// Mitsubishi GX Works2 project: BKVinaMainV1   PLC: FX3U/FX3UC

// global labels: Global1
VAR_GLOBAL
  RelayMXDT_1 AT Y002 : BOOL;
  RelayMXDT_2 AT Y006 : BOOL;
  RelayMXDP_1 AT Y003 : BOOL;
  RelayMXDP_2 AT Y007 : BOOL;
  RelayMQ_R AT Y010 : BOOL;
  MR_DSLOW AT Y011 : BOOL;
  RelayMR_1 AT Y012 : BOOL;
  RelayMR_2 AT Y013 : BOOL;
  RelayTT AT Y014 : BOOL;
  ALARM AT Y015 : BOOL;
  OPERATION AT Y016 : BOOL;
  RelayXLKC1 AT Y017 : BOOL;
  RelayXLC2 AT Y020 : BOOL;
  RelayXLD3_1 AT Y021 : BOOL;
  RelayXLD3_2 AT Y022 : BOOL;
  RelayXLX4_1 AT Y023 : BOOL;
  RelayXLX4_2 AT Y024 : BOOL;
  RelayXLX5_1 AT Y025 : BOOL;
  RelayXLX5_2 AT Y026 : BOOL;
  RelayXLD6_1 AT Y027 : BOOL;
  RelayXLD6_2 AT Y030 : BOOL;
  RelayXLTT AT Y031 : BOOL;
  RelayXLTP AT Y032 : BOOL;
  RelayXLKDT AT Y035 : BOOL;
  RelayLubOil AT Y036 : BOOL;
  RelayOilP AT Y037 : BOOL;
  RelayOilV1 AT Y040 : BOOL;
  RelayOilV2 AT Y041 : BOOL;
  CommandMXC_F : BOOL;
  CommandMXC_Z : BOOL;
  CommandMQ_F : BOOL;
  CommandMQ_Z : BOOL;
  CommandMXDT_F : BOOL;
  CommandMXDT_Z : BOOL;
  CommandMXDP_F : BOOL;
  CommandMXDP_Z : BOOL;
  CommandMR_L : BOOL;
  CommandMR_R : BOOL;
  CommandXLXC_I : BOOL;
  CommandXLXC_O : BOOL;
  MR_L AT X010 : BOOL;
  MR_R AT X011 : BOOL;
  CB3 AT X012 : BOOL;
  EMERG AT X013 : BOOL;
  MainRST AT X014 : BOOL;
  START AT X015 : BOOL;
  Jog_Left AT X016 : BOOL;
  Jog_Right AT X017 : BOOL;
  PushOilPump AT X020 : BOOL;
  XLKC1_I AT X021 : BOOL;
  XLKC1_O AT X022 : BOOL;
  XLC2_I AT X023 : BOOL;
  XLC2_O AT X024 : BOOL;
  XLD3_I AT X025 : BOOL;
  XLD3_O AT X026 : BOOL;
  XLX4_I AT X027 : BOOL;
  XLX4_O AT X030 : BOOL;
  XLX5_I AT X031 : BOOL;
  XLX5_O AT X032 : BOOL;
  XLD6_I AT X033 : BOOL;
  XLD6_O AT X034 : BOOL;
  XLTT_I AT X035 : BOOL;
  XLTP_I AT X036 : BOOL;
  XLTT_O AT X037 : BOOL;
  XLTP_O AT X040 : BOOL;
  XLDT_I AT X041 : BOOL;
  XLDT_O AT X042 : BOOL;
  XLDP_I AT X043 : BOOL;
  XLDP_O AT X044 : BOOL;
  OLPump AT X045 : BOOL;
  MR_L1 AT X046 : BOOL;
  MR_R1 AT X047 : BOOL;
  RelayMQ_2 AT Y005 : BOOL;
  RelayMXC_1 AT Y000 : BOOL;
  RelayMXC_2 AT Y004 : BOOL;
  RelayMQ_1 AT Y001 : BOOL;
  MXDT_ZX AT X002 : BOOL;
  MXDP_ZX AT X003 : BOOL;
  MXC_ZX AT X004 : BOOL;
  MQ_ZX AT X005 : BOOL;
  MXC_FWD : BOOL;
  MQ_FWD : BOOL;
  MXDT_FWD : BOOL;
  MXDP_FWD : BOOL;
  ModeAuto : BOOL;
  StopEmerg : BOOL;
  activeCK : BOOL;
  pushManXLKC1 AT M200 : BOOL;
  pushManXLC2 AT M201 : BOOL;
  pushManXLD3_I AT M202 : BOOL;
  pushManXLD3_O AT M203 : BOOL;
  pushManXLX4_I AT M204 : BOOL;
  pushManXLX4_O AT M205 : BOOL;
  pushManXLX5_I AT M206 : BOOL;
  pushManXLX5_O AT M207 : BOOL;
  pushManXLD6_I AT M208 : BOOL;
  pushManXLD6_O AT M209 : BOOL;
  pushManXLTT AT M210 : BOOL;
  pushManXLTP AT M211 : BOOL;
  pushManXLKDT AT M212 : BOOL;
  pushManXLKDP AT M213 : BOOL;
  pushManXLDT AT M214 : BOOL;
  pushManXLDP AT M215 : BOOL;
  pushManTT AT M216 : BOOL;
  pushManMXC_F AT M217 : BOOL;
  pushManMXC_Z AT M218 : BOOL;
  pushManMQ_F AT M219 : BOOL;
  pushManMQ_Z AT M220 : BOOL;
  pushManMXDT_F AT M221 : BOOL;
  pushManMXDT_Z AT M222 : BOOL;
  pushManMXDP_F AT M223 : BOOL;
  pushManMXDP_Z AT M224 : BOOL;
  PushOilV1 AT M225 : BOOL;
  PushOilV2 AT M226 : BOOL;
  pushB8 AT M227 : BOOL;
  pushB9 AT M228 : BOOL;
  pushB10 AT M229 : BOOL;
  pushCa1 AT M230 : BOOL;
  pushCa2 AT M231 : BOOL;
  pushCa3 AT M232 : BOOL;
  rstTotalB AT M233 : BOOL;
  rstCounterCK AT M234 : BOOL;
  rstAmountCK AT M235 : BOOL;
  restory AT M236 : BOOL;
  PushLubOil AT M237 : BOOL;
  PushPause AT M238 : BOOL;
  Pape0 AT M239 : BOOL;
  Pape1 AT M240 : BOOL;
  Pape2 AT M241 : BOOL;
  Pape3 AT M242 : BOOL;
  CommandXLX5_I : BOOL;
  CommandXLX5_O : BOOL;
  CommandXLXD_I : BOOL;
  CommandXLXD_O : BOOL;
  CommandXLD6_I : BOOL;
  PauseAlarm AT M243 : BOOL;
  RelayXLDT AT Y033 : BOOL;
  RelayXLDP AT Y034 : BOOL;
  PauseMR AT M244 : BOOL;
  Real_MXC : REAL;
  Real_MQ : REAL;
  Real_MXDT : REAL;
  Real_MXDP : REAL;
  Counter_MQ : DINT;
  Round_MXC AT D200 : REAL;
  Round_MQL AT D202 : REAL;
  Round_MQR AT D204 : REAL;
  Round_MXDT AT D206 : REAL;
  Round_MXDP AT D208 : REAL;
  IndicateMXC AT D210 : REAL;
  IndicateMQ AT D212 : REAL;
  IndicateMXDT AT D214 : REAL;
  IndicateMXDP AT D216 : REAL;
  NumberCK AT D220 : DWORD;
  CounterCK AT D222 : DWORD;
  AmountCK AT D224 : DWORD;
  TotalCK AT D226 : DWORD;
  rstPauseMR AT M245 : BOOL;
  ca1_B8 AT D250 : DWORD;
  ca2_B8 AT D252 : DWORD;
  ca3_B8 AT D254 : DWORD;
  ca1_B9 AT D256 : DWORD;
  ca2_B9 AT D258 : DWORD;
  ca3_B9 AT D260 : DWORD;
  ca1_B10 AT D262 : DWORD;
  ca2_B10 AT D264 : DWORD;
  ca3_B10 AT D266 : DWORD;
  total_B8 AT D268 : DWORD;
  total_B9 AT D270 : DWORD;
  total_B10 AT D272 : DWORD;
  CommandMXDT : BOOL;
  CommandMXDP : BOOL;
  CommandBTX : BOOL;
  CommandXLTT : BOOL;
  CommandXLTP : BOOL;
  CommandXLDT : BOOL;
  CommandXLDP : BOOL;
  CommandXLKDT : BOOL;
  CommandXLKDP : BOOL;
  CommandXLKC1 : BOOL;
  MXC_Z : BOOL;
  MQ_Z : BOOL;
  MXDT_Z : BOOL;
  MXDP_Z : BOOL;
  MQ_LimitF : BOOL;
  MQ_LimitR : BOOL;
  CommandXLD6_O : BOOL;
  TimeMR_DSL AT D230 : DWORD;
  TimeMQ_Z AT D232 : DWORD;
  TimeMR_E AT D234 : DWORD;
  TimeERROR AT D236 : DWORD;
  TimeMXD AT D238 : DWORD;
END_VAR

// task InterruptMQ_Z (event I501, interval 0, priority 31): PickupX005
// task InterruptMXC (event I010, interval 0, priority 31): EncoderX001
// task InterruptMXC_Z (event I401, interval 0, priority 31): PickupX004
// task InterruptMXDP (event I030, interval 0, priority 31): EncoderX007
// task InterruptMXDP_Z (event I301, interval 0, priority 31): PickupX003
// task InterruptMXDT (event I020, interval 0, priority 31): EncoderX006
// task InterruptMXDT_Z (event I201, interval 0, priority 31): PickupX002
// task Task_01 (event TRUE, interval 0, priority 31): PowerControl, StepControl

PROGRAM EncoderX001
SET( TRUE , MXC_FWD );
SET( TRUE, CommandMXC_Z);
RST( TRUE, CommandXLXC_O);
RST( TRUE, CommandXLXD_O);
END_PROGRAM

PROGRAM EncoderX006
SET( TRUE , MXDT_FWD );
RST( TRUE, CommandXLDT);
RST( TRUE, CommandMXDT_F);
RST( TRUE, CommandMXDT);
SET( XLX4_O AND activeCK, CommandXLXC_I); 
SET( XLD3_O AND activeCK, CommandXLXD_I);
END_PROGRAM

PROGRAM EncoderX007
SET( TRUE , MXDP_FWD );
RST( TRUE, CommandXLDP);
RST( TRUE, CommandMXDP_F);
RST( TRUE, CommandMXDP);
END_PROGRAM

FUNCTION_BLOCK MotorOne
VAR_INPUT
  SetAutoMan : BOOL;
  PushMan : BOOL;
  LimitInput : BOOL;
END_VAR
VAR_IN_OUT
  SetAutoRun : BOOL;
END_VAR
VAR_OUTPUT
  Output : BOOL;
END_VAR
VAR
  RelayBuffer : BOOL;
END_VAR
(* Set mode Auto / Mannual *)
IF  SetAutoMan THEN
	RelayBuffer := SetAutoRun;
ELSE 
	RelayBuffer := PushMan;
END_IF;

Output := RelayBuffer AND NOT LimitInput ;
(* Reset control signal *)
RST(LDP(TRUE, LimitInput), SetAutoRun );
END_FUNCTION_BLOCK

FUNCTION_BLOCK MotorRev
VAR_INPUT
  SetAutoMan : BOOL;
END_VAR
VAR_IN_OUT
  PushManF : BOOL;
  PushManR : BOOL;
END_VAR
VAR_INPUT
  LimitInputF : BOOL;
  LimitInputR : BOOL;
END_VAR
VAR_IN_OUT
  SetAutoRunF : BOOL;
  SetAutoRunR : BOOL;
END_VAR
VAR_OUTPUT
  OutputF : BOOL;
  OutputR : BOOL;
END_VAR
VAR
  RelayBufferF : BOOL;
  RelayBufferR : BOOL;
END_VAR
(* Set mode Auto/Man *)
IF  SetAutoMan THEN
	RelayBufferF := 	NOT SetAutoRunR AND SetAutoRunF;
	RelayBufferR := NOT SetAutoRunF AND SetAutoRunR;
ELSE
	RelayBufferF := NOT PushManR AND PushManF;
	RelayBufferR := NOT PushManF AND PushManR;
END_IF;

OutputF := RelayBufferF AND NOT LimitInputF ;
OutputR := RelayBufferR AND NOT LimitInputR ;
(* Reset control signal *)
RST( LDP(TRUE, LimitInputF), SetAutoRunF );
RST( LDP(TRUE, LimitInputR), SetAutoRunR );
END_FUNCTION_BLOCK

PROGRAM PickupX002
SET(TRUE, MXDT_Z);
SET( TRUE, M8052);
RST( TRUE, CommandMXDT);
END_PROGRAM

PROGRAM PickupX003
SET(TRUE, MXDP_Z);
SET( TRUE, M8053);
RST( TRUE, CommandMXDP);
END_PROGRAM

PROGRAM PickupX004
SET( TRUE, MXC_Z);
SET( XLD3_O, CommandXLXD_I);
SET( XLX4_O, CommandXLXC_I);
SET( TRUE, M8054);
END_PROGRAM

PROGRAM PickupX005
DADD( MQ_LimitF, Counter_MQ, K1 , Counter_MQ);
SET( Counter_MQ >= REAL_TO_DINT( Real_MQ), MQ_FWD);
SET( MQ_LimitR , MQ_Z);
END_PROGRAM

PROGRAM PowerControl
VAR
  MR : MotorRev;
  MQ : MotorRev;
  MXC : MotorRev;
  MXDT : MotorRev;
  MXDP : MotorRev;
  XLKC1 : MotorOne;
  XLC2 : MotorOne;
  XLD3 : MotorRev;
  XLX4 : MotorRev;
  XLX5 : MotorRev;
  XLD6 : MotorRev;
  XLTT : MotorOne;
  XLTP : MotorOne;
  XLKDT : MotorOne;
  XLKDP : MotorOne;
  XLDT : MotorOne;
  XLDP : MotorOne;
  OILPUMP : MotorOne;
  VALVE1 : MotorOne;
  VALVE2 : MotorOne;
  ManualMXC_F : BOOL;
  ManualMXC_Z : BOOL;
  ManualMQ_F : BOOL;
  ManualMQ_Z : BOOL;
  ManualMXDT_F : BOOL;
  ManualMXDT_Z : BOOL;
  ManualMXDP_F : BOOL;
  ManualMXDP_Z : BOOL;
  CommandXLC2 : BOOL;
  ButtonOilP : BOOL;
  ButtonOilV1 : BOOL;
  ButtonOilV2 : BOOL;
  TimerMRDSL_Q : BOOL;
  TimerMQ_ZQ : BOOL;
  TimerMR_DSL : TON;
  TimerMQ_Z : TON;
  Dint_C251 : DINT;
  Dint_C234 : DINT;
  Dint_C244 : DINT;
  Dint_C245 : DINT;
  ManualXLD6 : BOOL;
  ManualXLDT : BOOL;
  ManualXLDP : BOOL;
  ManualXLKDT : BOOL;
  ManualXLKDP : BOOL;
  ManualXLX5_O : BOOL;
  ManualXLX5_I : BOOL;
  TimerXLTT : TON;
  TimerXLTP : TON;
  TimerXLTT_Q : BOOL;
  TimerXLTP_Q : BOOL;
END_VAR
EI( TRUE );
(* MR: Chạy khi cụm xoắn đầu chạy *)
MR(SetAutoMan := ModeAuto, PushManF := Jog_Left , PushManR := Jog_Right ,
		LimitInputF := MR_L, LimitInputR := MR_R,
		SetAutoRunF := CommandMR_L, SetAutoRunR := CommandMR_R ,
		OutputF := RelayMR_1, OutputR:= RelayMR_2);

RelayTT := (RelayMR_1 AND NOT MR_L) OR (RelayMR_2 AND NOT MR_R);
TimerMR_DSL(IN := (NOT MR_L AND RelayMR_1) OR (NOT MR_R AND RelayMR_2), 
								PT := DWORD_TO_TIME(TimeMR_DSL)/100, Q := TimerMRDSL_Q );
								
SET(LDP(TRUE, (MR_L1 AND RelayMR_1) OR (MR_R1 AND RelayMR_2)), MR_DSLOW);
RST(LDP(TRUE, (MR_L AND RelayMR_2) OR (MR_R AND RelayMR_1)), MR_DSLOW);

(* MXQ: *)	
SET(LDP(TRUE, MR_L OR MR_R), CommandMQ_F);
SET(LDP(TRUE, MR_L), RelayMQ_R);
RST(LDP(TRUE,MR_R), RelayMQ_R);
MQ(SetAutoMan := ModeAuto,
		PushManF := pushManMQ_F, PushManR := ManualMQ_Z,
		LimitInputF := MQ_FWD, LimitInputR := MQ_Z,
		SetAutoRunF := CommandMQ_F, SetAutoRunR := CommandMQ_Z, 
		OutputF := MQ_LimitF, OutputR:= MQ_LimitR);

IF RelayMQ_R THEN
	RelayMQ_1 := MQ_LimitF;
	RelayMQ_2 := MQ_LimitR;
ELSE
	RelayMQ_1 := MQ_LimitR;
	RelayMQ_2 := MQ_LimitF;
END_IF;
	
(* MXC:  CommandXLXC_I  and CommandXLXC_O *)	
MXC(SetAutoMan:= ModeAuto, 
			PushManF := pushManMXC_F, PushManR := ManualMXC_Z,
			LimitInputF := MXC_FWD, LimitInputR := MXC_Z,
			SetAutoRunF := CommandMXC_F, SetAutoRunR := CommandMXC_Z,
			OutputF := RelayMXC_1, OutputR := RelayMXC_2);

XLD3(SetAutoMan := ModeAuto,
			PushManF := pushManXLD3_O, PushManR := pushManXLD3_I,
			LimitInputF := XLD3_O, LimitInputR := XLD3_I,
			SetAutoRunF := CommandXLXD_O, SetAutoRunR := CommandXLXD_I,
			OutputF := RelayXLD3_1, OutputR := RelayXLD3_2);			
			
XLX4(SetAutoMan := ModeAuto,
			PushManF := pushManXLX4_O, PushManR := pushManXLX4_I,
			LimitInputF := XLX4_O , LimitInputR := XLX4_I,
			SetAutoRunF := CommandXLXC_O, SetAutoRunR := CommandXLXC_I,
			OutputF := RelayXLX4_1, OutputR := RelayXLX4_2);				

(* PHA:  CommandPHA_1  and CommandPHA_2 *)	
XLX5(SetAutoMan := ModeAuto,
			PushManF := pushManXLX5_O, PushManR := pushManXLX5_I,
			LimitInputF := NOT XLX4_I OR XLX5_O, LimitInputR := NOT XLX4_I OR XLX5_I,
			SetAutoRunF := CommandXLX5_O, SetAutoRunR := CommandXLX5_I,
			OutputF := RelayXLX5_1, OutputR := RelayXLX5_2);			

XLD6(SetAutoMan := ModeAuto,
			PushManF := pushManXLD6_O, PushManR := pushManXLD6_I,
			LimitInputF := FALSE, LimitInputR := FALSE,
			SetAutoRunF := CommandXLD6_O, SetAutoRunR := CommandXLD6_I, 
			OutputF := RelayXLD6_1, OutputR := RelayXLD6_2);				

(* MXDT:  CommandXLDT => dừng khi encoder đủ vòng *)	
SET( LDP(TRUE,  XLDT_I), CommandMXDT_Z);
MXDT(SetAutoMan := ModeAuto, 
			PushManF := pushManMXDT_F,  PushManR := ManualMXDT_Z,
			LimitInputF := MXDT_FWD, LimitInputR := MXDT_Z,
			SetAutoRunF :=  CommandMXDT_F, SetAutoRunR := CommandMXDT_Z ,
			OutputF := RelayMXDT_1, OutputR := RelayMXDT_2);

ManualXLDT := LDP(TRUE, pushManXLDT) XOR ManualXLDT;
RST( ModeAuto, ManualXLDT);
RelayXLDT := CommandXLDT OR ManualXLDT;

(* MXDP:  CommandXLDP => dừng khi encoder đủ vòng *)	
SET( LDP(TRUE, XLDP_I), CommandMXDP_Z);
MXDP(SetAutoMan := ModeAuto, 
			PushManF := pushManMXDP_F, PushManR := ManualMXDP_Z,
			LimitInputF := MXDP_FWD, LimitInputR := MXDP_Z,
			SetAutoRunF := CommandMXDP_F, SetAutoRunR := CommandMXDP_Z ,
			OutputF := RelayMXDP_1, OutputR := RelayMXDP_2);
			
ManualXLDP := LDP(TRUE, pushManXLDP) XOR ManualXLDP;
RST( ModeAuto, ManualXLDP);		
RelayXLDP := CommandXLDP OR ManualXLDP;

(* BTX:  CommandBTX  *)
RST(LDP(TRUE, CommandBTX AND XLKC1_O AND RelayXLKC1), CommandXLKC1);
SET(LDP(TRUE, CommandBTX AND XLC2_O AND RelayXLC2), CommandXLKC1);

RelayXLKC1 := (CommandXLKC1 AND ModeAuto) OR pushManXLKC1;

SET(LDP(TRUE, NOT XLKC1_O AND XLKC1_I), CommandXLC2);
RST(LDP(TRUE, NOT XLKC1_I AND XLKC1_O), CommandXLC2);
RST(LDP(TRUE, NOT XLKC1_I AND XLKC1_O), CommandBTX);

RelayXLC2 := (CommandXLC2 AND ModeAuto) OR pushManXLC2;

(* TLT: CommandXLTT => chạy theo cylinder  xoắn đầu *)
RelayXLTT := (RelayMXDT_1 AND ModeAuto) OR pushManXLTT;

(* TLP: CommandXLTP => chạy theo cylinder  xoắn đầu *)
RelayXLTP := (RelayMXDP_1 AND ModeAuto) OR pushManXLTP;

(* Hydrolic control *)
ButtonOilP := LDP(TRUE, PushOilPump) XOR ButtonOilP;
OILPUMP(PushMan := ButtonOilP, LimitInput := OLPump, Output := RelayOilP );

RelayOilV1 := RelayMQ_1 OR RelayMQ_2 OR RelayMXDP_1 OR RelayMXDP_2 
OR RelayMXDT_1 OR RelayMXDT_2 OR RelayXLX5_1 OR RelayXLX5_2;
RelayOilV2 := RelayMXC_1 OR RelayMXC_2 OR RelayXLD3_1 
OR RelayXLD3_2 OR RelayXLX4_1 OR RelayXLX4_2;
RelayLubOil := LDP(TRUE, PushLubOil) XOR RelayLubOil;

IF ModeAuto THEN
	(* Forward at Zero *)
	RST( CommandMXC_F AND MXC_ZX, MXC_FWD);
	RST( CommandMQ_F AND MQ_ZX, MQ_FWD);
	RST( CommandMXDT_F AND MXDT_ZX, MXDT_FWD);
	RST( CommandMXDP_F AND MXDP_ZX, MXDP_FWD);
	
	(* Set Home *)
	RST( LDP(TRUE, CommandMXC_Z), MXC_Z);
	RST( LDP(TRUE, CommandMQ_Z), MQ_Z);
	RST( LDP(TRUE, CommandMXDT_Z), MXDT_Z);
	RST( LDP(TRUE, CommandMXDP_Z), MXDP_Z);

ELSE	
	RST( LDP(TRUE, pushManMXC_F), MXC_FWD);
	RST( LDP(TRUE, pushManMQ_F), MQ_FWD);
	RST( LDP(TRUE, pushManMXDT_F), MXDT_FWD);
	RST( LDP(TRUE, pushManMXDP_F), MXDP_FWD);
	
	SET( LDP(TRUE, pushManMXC_Z), ManualMXC_Z);
	SET( LDP(TRUE, pushManMQ_Z), ManualMQ_Z);
	SET( LDP(TRUE, pushManMXDT_Z), ManualMXDT_Z);
	SET( LDP(TRUE, pushManMXDP_Z), ManualMXDP_Z);
	
	RST( LDP(TRUE, ManualMXC_Z), MXC_Z);
	RST( LDP(TRUE, ManualMQ_Z), MQ_Z);
	RST( LDP(TRUE, ManualMXDT_Z), MXDT_Z);
	RST( LDP(TRUE, ManualMXDP_Z), MXDP_Z);
	
	RST( LDP(TRUE, MXC_Z), ManualMXC_Z);
	RST( LDP(TRUE, MQ_Z), ManualMQ_Z);
	RST( LDP(TRUE, MXDT_Z), ManualMXDT_Z);
	RST( LDP(TRUE, MXDP_Z), ManualMXDP_Z);
	
	(* initialize encoder interrupt *)
	DMOVP( pushManMXC_F, 0, C251);
	DMOVP( pushManMQ_F, 0, Counter_MQ);
	DMOVP( pushManMXDT_F, 0, C244);
	DMOVP( pushManMXDP_F, 0, C245);
END_IF;

DWORD_TO_DINT_E( TRUE , C251 , Dint_C251 );
DWORD_TO_DINT_E( TRUE , C244 , Dint_C244 );
DWORD_TO_DINT_E( TRUE , C245 , Dint_C245 );

DEDIV( TRUE , DINT_TO_REAL(Dint_C251) , 2000.0 , IndicateMXC);
DEDIV( TRUE , DINT_TO_REAL(Counter_MQ) , 2.0 , IndicateMQ);
DEDIV( TRUE , DINT_TO_REAL(Dint_C244) , 360.0 , IndicateMXDT);
DEDIV( TRUE , DINT_TO_REAL(Dint_C245) , 360.0 , IndicateMXDP);

(* Set Interrupt *)
RST( LDP(TRUE, RelayMXC_2), M8054);
RST( RelayMQ_1 OR RelayMQ_2, M8055);
RST( LDP(TRUE, RelayMXDT_2), M8052);
RST( LDP(TRUE, RelayMXDP_2), M8053);

(* initialize encoder interrupt *)
DMOVP( CommandMXC_F, 0, C251);
DMOVP( CommandMQ_F, 0, Counter_MQ);
DMOVP( CommandMXDT_F, 0, C244);
DMOVP( CommandMXDP_F, 0, C245);

M8390 := M8388;
M8391 := M8388;
(*đảo chiều counter*)
M8244 := RelayMXDT_2;
M8245 := RelayMXDP_2;

(* Initialize high speed counter *)
OUT_C_32( TRUE, CC251, K2147483647);
OUT_C_32( TRUE, CC244, K2147483647);
OUT_C_32( TRUE, CC245, K2147483647);

(* Initialize high speed counter *)
DHSCS_I( TRUE , REAL_TO_DINT( Real_MXC ), CN251, I010);
DHSCS_I( TRUE , REAL_TO_DINT( Real_MXDT ), CN244, I020);
DHSCS_I( TRUE , REAL_TO_DINT( Real_MXDP ), CN245, I030);
END_PROGRAM

FUNCTION_BLOCK Servo
VAR_INPUT
  SetAutoMan : BOOL;
END_VAR
VAR_IN_OUT
  PushManF : BOOL;
  PushManR : BOOL;
END_VAR
VAR_INPUT
  Speed : DWORD;
  Range : DWORD;
END_VAR
VAR_IN_OUT
  SetAutoRunF : BOOL;
  SetAutoRunR : BOOL;
END_VAR
VAR_OUTPUT
  OutputPLS : BOOL;
  OutputDIR : BOOL;
END_VAR
VAR
  RelayPLS : BOOL;
  RelayDIR : BOOL;
END_VAR
VAR_INPUT
  LimitInputF : BOOL;
  LimitInputR : BOOL;
END_VAR
(* Set mode Auto/Man *)
IF  SetAutoMan THEN
	RelayDIR := SetAutoRunR;
	RelayPLS := SetAutoRunF XOR SetAutoRunR;
ELSE
	RelayDIR := PushManR;
	RelayPLS := PushManF XOR PushManR;
END_IF;

OutputDIR := RelayDIR ;

DPLSY( RelayPLS , Speed, Range , OutputPLS );

(* Reset control signal *)
RST( LDF( TRUE, LimitInputF ) , SetAutoRunF );
RST( LDF( TRUE, LimitInputR ) , SetAutoRunR );
END_FUNCTION_BLOCK

PROGRAM StepControl
VAR
  FistScan : BOOL;
  Emergency : BOOL;
  AutoEnable : BOOL;
  AuxCylinder : BOOL;
  MainCylinder : BOOL;
  TimerRestore : TON;
  TimerMR_E : TON;
  TimerERROR : TON;
  TimerMXDT : TON;
  TimerMXDP : TON;
  rstCa : BOOL;
  Error : ARRAY [0..18] OF BOOL;
  status : ARRAY [0..9] OF BOOL;
  cond : ARRAY [0..9] OF BOOL;
  count : INT;
  TimerMRR_Q : BOOL;
  TimerMRE_Q : BOOL;
  TimerERROR_Q : BOOL;
  TimerRestore_Q : BOOL;
  TimerMXDT_Q : BOOL;
  TimerMXDP_Q : BOOL;
  CylinderPha1 : BOOL;
  CylinderPha2 : BOOL;
  pointer : INT;
END_VAR
(*
Thake production line project: Mr. Chim Van Cang - Mr. Nguyen Tuan Nam
Code and graphic designer: HadiMadu - Techwaves Co,.Ltd
*)
Emergency := EMERG;

ALARM :=  NOT AutoEnable OR PauseAlarm;

SET(LDP(TRUE, MainRST), AutoEnable);
RST(LDP(TRUE, Emergency AND START), pointer);
SET(LDP(TRUE, Emergency AND START), status[0]);
RST(LDP(TRUE, Emergency AND START), AutoEnable);	

SET(LDP(TRUE, TimerMRE_Q), PauseMR);
RST(LDP(TRUE, rstPauseMR), PauseMR);

PauseAlarm := NOT CB3 OR PushPause OR PauseMR OR OLPump OR Emergency;(*OR TimerERROR_Q*)

OPERATION := status[1] OR status[2] OR status[3] OR status[4] OR status[5] OR status[6];
(* Mode Auto *)
ModeAuto := AutoEnable AND NOT PauseAlarm;

Pape0 := NOT ModeAuto;
Pape1 := status[0] OR status[1] OR status[2];
Pape2 := status[3] OR status[4];
Pape3 := status[5] OR status[6];

(* Power control *)
AuxCylinder := XLTT_I AND XLTP_I; 
MainCylinder := XLD3_I AND XLX4_I AND XLDT_I AND XLDP_I AND MQ_ZX;
CylinderPha1 := MR_L AND XLD6_O AND XLX5_I AND MXDT_ZX;
CylinderPha2 := MR_R AND XLD6_I AND XLX5_O AND MXDP_ZX;

cond[0] := pointer = 0 AND ModeAuto AND CylinderPha1 AND MainCylinder AND START; 			(* S1: Điều kiện chạy MQ*)
cond[1] := pointer = 1 AND ModeAuto AND LDP(TRUE, MQ_FWD AND MainCylinder AND AuxCylinder); 		(* S2: Điều kiện chạy BXT*)
cond[2] := pointer = 2 AND ModeAuto AND LDP(TRUE, XLKC1_O);  						(* S3: Điều kiện chạy MXDT, MR-L*)
cond[3] := pointer = 3 AND ModeAuto AND LDP(TRUE, MQ_FWD AND MainCylinder AND AuxCylinder);  		(* S4: Điều kiện chạy BXT, PHA 2*)
cond[4] := pointer = 4 AND ModeAuto AND LDP(TRUE, CylinderPha2 AND MainCylinder AND XLKC1_O); 		(* S5: Điều kiện chạy MXDT, MR-R*)
cond[5] := pointer = 5 AND ModeAuto AND LDP(TRUE, MQ_FWD AND MainCylinder AND AuxCylinder); 		(* S6: Điều kiện chạy BXT, PHA 1*)
cond[6] := pointer = 6 AND ModeAuto AND LDP(TRUE, CylinderPha1 AND MainCylinder AND XLKC1_O); 		(* S3: Điều kiện chạy MXDP, MR-L*)

(*cycle control*)
SET( LDP( TRUE, status[1]), CommandMQ_F);
SET( LDP( TRUE, status[2] OR status[4] OR status[6]), CommandBTX); 
SET( LDP( TRUE, status[4]), CommandXLX5_O);		
RST( LDP( TRUE, status[4]), CommandXLD6_O);	
SET( LDP( TRUE, status[4]), CommandXLD6_I);
SET( LDP( TRUE, status[6]), CommandXLX5_I); 	
RST( LDP( TRUE, status[6]), CommandXLD6_I);		
SET( LDP( TRUE, status[6]), CommandXLD6_O);	

SET( LDP( TRUE, status[5] OR status[3]), CommandXLXC_O);     
SET( LDP( TRUE, status[5] OR status[3]), CommandXLXD_O);

SET( LDP(TRUE, NOT activeCK AND XLD3_O AND XLX4_O), CommandMXC_F);

SET( LDP(TRUE, status[3]), CommandXLDT); 
SET( LDP(TRUE, status[5]), CommandXLDP);

SET( LDP(TRUE, NOT CommandMXDT_F AND XLX4_O AND XLDT_O AND status[3]), CommandMXDT);
SET( LDP(TRUE, NOT CommandMXDP_F AND XLX4_O AND XLDP_O AND status[5]), CommandMXDP);
TimerMXDT( IN := CommandMXDT, 	PT := DWORD_TO_TIME( TimeMXD), Q := TimerMXDT_Q);
TimerMXDP( IN := CommandMXDP, 	PT := DWORD_TO_TIME( TimeMXD), Q := TimerMXDP_Q);					
SET( LDP(TRUE, TimerMXDT_Q OR pushManMXDT_F), CommandMXDT_F);
SET( LDP(TRUE, TimerMXDP_Q OR pushManMXDP_F), CommandMXDP_F);

SET(LDP(TRUE, NOT MR_L AND MR_R AND status[5]), CommandMR_L);
SET(LDP(TRUE, NOT MR_R AND MR_L AND status[3]), CommandMR_R);
TimerMR_E( IN := RelayMR_1 OR RelayMR_2,
						PT := DWORD_TO_TIME( TimeMR_E) *1000, Q := TimerMRE_Q);						

(*Control status 0*)  
RST(LDP(TRUE, status[0]), CommandMR_R);
RST(LDP(TRUE, status[0]), CommandMR_L);
RST(LDP(TRUE, Status[0]), CommandMXC_F);
RST(LDP(TRUE, Status[0]), CommandMXC_Z);
RST(LDP(TRUE, Status[0]), CommandMQ_F);
RST(LDP(TRUE, Status[0]), CommandMQ_Z);
RST(LDP(TRUE, Status[0]), CommandMXDT_F);
RST(LDP(TRUE, Status[0]), CommandMXDT_Z);
RST(LDP(TRUE, Status[0]), CommandMXDP_F);
RST(LDP(TRUE, Status[0]), CommandMXDP_Z);
RST(Status[0], CommandXLXC_O);
RST(Status[0], CommandXLXD_O);
RST(LDP(TRUE, Status[0]), CommandXLXC_I);
RST(LDP(TRUE, Status[0]), CommandXLXD_I);
RST(LDP(TRUE, Status[0]), CommandXLX5_I);   
RST(LDP(TRUE, Status[0]), CommandXLD6_I); 
RST(LDP(TRUE, Status[0]), CommandXLX5_O); 
RST(LDP(TRUE, Status[0]), CommandXLD6_O);
RST(LDP(TRUE, Status[0]), CommandXLDT); 
RST(LDP(TRUE, Status[0]), CommandXLDP);
RST(LDP(TRUE, Status[0]), CommandBTX);
RST(LDP(TRUE, Status[0]), CommandXLKC1);
RST(Status[0], CommandXLTT); 
RST(Status[0], CommandXLTP);

SET(LDP(TRUE, NOT MR_L AND ModeAuto AND MainRST), CommandMR_L);
SET(LDP(TRUE, NOT MXC_ZX AND ModeAuto AND MainRST), CommandMXC_Z);
SET(LDP(TRUE, NOT MQ_ZX AND ModeAuto AND MainRST), CommandMQ_Z);
SET(LDP(TRUE, NOT MXDT_ZX AND ModeAuto AND MainRST), CommandMXDT_Z);
SET(LDP(TRUE, NOT MXDP_ZX AND ModeAuto AND MainRST), CommandMXDP_Z);
SET(LDP(TRUE, NOT XLX4_I AND ModeAuto AND MainRST), CommandXLXC_I); 
SET(LDP(TRUE, NOT XLD3_I AND ModeAuto AND MainRST), CommandXLXD_I); 
SET(LDP(TRUE, NOT XLX5_I AND XLX4_I AND ModeAuto AND MainRST), CommandXLX5_I); 
SET(LDP(TRUE, NOT XLD6_O AND XLD3_I AND ModeAuto AND MainRST), CommandXLD6_O);
	
(*cycle program*)
IF ModeAuto THEN 
	FOR count := 0 TO 6 DO
		IF (count = 0) AND cond[0] THEN
			pointer := 1;
			status[pointer] := 1;
		END_IF;
		IF (count = 1) AND cond[1] THEN
			pointer := 2;
			status[pointer] := 1;
		END_IF;
		IF (count = 2) AND cond[2] THEN
			pointer := 3;
			status[pointer] := 1;
		END_IF;
		IF (count = 3) AND cond[3] THEN
			pointer := 4;
			status[pointer] := 1;
		END_IF;
		IF (count = 4) AND cond[4] THEN
			pointer := 5;
			status[pointer] := 1;
		END_IF;
		IF (count = 5) AND cond[5] THEN
			pointer := 6;
			status[pointer] := 1;
		END_IF;
		IF (count = 6) AND cond[6] THEN
			pointer := 3;
			status[pointer] := 1;
		END_IF;
		IF (count <> pointer) THEN
			status[count] := 0;
		END_IF;				
	END_FOR;
END_IF;

Error[0] := Error[1] OR Error[2] OR Error[3] OR Error[4] OR Error[5] OR Error[6] OR Error[7] OR Error[8] OR Error[9]
 					OR Error[10] OR Error[11] OR Error[12] OR Error[13] OR Error[14] OR Error[15] OR Error[16];
 					
TimerERROR(IN := Error[0], PT := DWORD_TO_TIME( TimeERROR)*1000, Q := TimerERROR_Q);

Error[1] := (RelayXLKC1 AND XLKC1_I) OR (RelayXLKC1 AND NOT XLKC1_O) OR (XLKC1_I AND XLKC1_O);
Error[2] := (RelayXLC2 AND XLC2_I) OR (RelayXLC2 AND NOT XLC2_O) OR (XLC2_I AND XLC2_O);
Error[3] := (RelayXLD3_1 AND XLD3_I) OR (RelayXLD3_2 AND XLD3_O) OR (XLD3_I AND XLD3_O);
Error[4] := (RelayXLX4_1 AND XLX4_I) OR (RelayXLX4_2 AND XLX4_O) OR (XLX4_I AND XLX4_O);
Error[5] := (RelayXLX5_1 AND XLX5_I) OR (RelayXLX5_2 AND XLX5_O) OR (XLX5_I AND XLX5_O);
Error[6] := (RelayXLD6_1 AND XLD6_I) OR (NOT RelayXLD6_1 AND XLD6_O) OR (XLD6_I AND XLD6_O);
Error[7] := (RelayXLDT AND XLDT_I) OR (RelayXLDT AND NOT XLDT_O) OR (XLDT_I AND XLDT_O);
Error[8] := (RelayXLDP AND XLDP_I) OR (RelayXLDP AND NOT XLDP_O) OR (XLDP_I AND XLDP_O);

Error[11] := (RelayXLTT AND XLTT_I);
Error[12] := (RelayXLTP AND XLTP_I);
Error[13] := NOT CommandMQ_Z AND MQ_ZX;
Error[14] := NOT CommandMXC_Z AND MXC_ZX;
Error[15] := NOT CommandMXDT_Z AND MXDT_ZX;
Error[16] := NOT CommandMXDP_Z AND MXDP_ZX;

TimerRestore(IN := restory, PT:= T#10s, Q := TimerRestore_Q);
IF TimerRestore_Q THEN
	Round_MQL := 1.5;
	Round_MQR := 1.5;
	Round_MXC := 2.05;
	Round_MXDT := 2.1;
	Round_MXDP := 2.1;
	NumberCK := 44;
	TimeERROR := 10;
	TimeMR_DSL := 200;
	TimeMXD := 600;
	TimeMR_E := 10;
END_IF;

(* Khai bao vong quay cho MXC *)
DEMUL( TRUE, E2000.0, Round_MXC , Real_MXC);
(* Khai báo vòng quay cho MQ bên trái *)
DEMUL( MR_L, E2.0, Round_MQL , Real_MQ);
(* Khai báo vòng quay cho MQ bên phải *)
DEMUL( MR_R, E2.0, Round_MQR , Real_MQ);
(* Khai báo vòng quay cho MXDT *)
DEMUL( TRUE, E360.0, Round_MXDT , Real_MXDT);
(* Khai báo vòng quay cho MXDP *)
DEMUL( TRUE, E360.0, Round_MXDP , Real_MXDP);

(* Khai bao thống kê sản lượng *)
DINCP( status[3] AND XLKC1_O, CounterCK);
activeCK := CounterCK >= NumberCK;
	
DINCP( pushB8 AND pushCa1 AND activeCK, ca1_B8 );
DINCP( pushB9 AND pushCa1 AND activeCK, ca1_B9 );
DINCP( pushB10 AND pushCa1 AND activeCK, ca1_B10 );
DINCP( pushB8 AND pushCa2 AND activeCK, ca2_B8 );
DINCP( pushB9 AND pushCa2 AND activeCK, ca2_B9 );
DINCP( pushB10 AND pushCa2 AND activeCK, ca2_B10 );
DINCP( pushB8 AND pushCa3 AND activeCK, ca3_B8 );
DINCP( pushB9 AND pushCa3 AND activeCK, ca3_B9 );
DINCP( pushB10 AND pushCa3 AND activeCK, ca3_B10 );
DINCP( pushB8 AND activeCK, total_B8 );
DINCP( pushB9 AND activeCK, total_B9 );
DINCP( pushB10 AND activeCK, total_B10 );

DINCP( activeCK, TotalCK);
DINCP( activeCK AND (pushCa1 OR pushCa2 OR pushCa3), AmountCK);
RST( rstCounterCK OR status[4] AND activeCK, CounterCK );
RST( LDF(TRUE, pushCa1 OR pushCa2 OR pushCa3), AmountCK);
RST(rstAmountCK, TotalCK);


IF rstTotalB THEN
	ca1_B8 := 0;
	ca1_B9 := 0;
	ca1_B10 := 0;
	ca2_B8 := 0;
	ca2_B9 := 0;
	ca2_B10 := 0;
	ca3_B8 := 0;
	ca3_B9 := 0;
	ca3_B10 := 0;
	total_B8 := 0;
	total_B9 := 0;
	total_B10 := 0;
END_IF;

RST(LDP(TRUE, pushB8), pushB9);
RST(LDP(TRUE, pushB8), pushB10);
RST(LDP(TRUE, pushB9), pushB8);
RST(LDP(TRUE, pushB9), pushB10);
RST(LDP(TRUE, pushB10), pushB8);
RST(LDP(TRUE, pushB10), pushB9);

RST(LDP(TRUE, pushCa1), pushCa2);
RST(LDP(TRUE, pushCa1), pushCa3);
RST(LDP(TRUE, pushCa2), pushCa1);
RST(LDP(TRUE, pushCa2), pushCa3);
RST(LDP(TRUE, pushCa3), pushCa1);
RST(LDP(TRUE, pushCa3), pushCa2);
END_PROGRAM
